// TIA Portal V16 export
// export: Created 2022-02-04T14:40:09.9916487Z, ExportSetting WithDefaults, DisplayName Totally Integrated Automation Portal, DisplayVersion V16 Update 1, DisplayName TIA Portal Version Control Interface, DisplayVersion V16, DisplayName TIA Portal Openness, DisplayVersion V16, DisplayName SINAMICS Startdrive Advanced, DisplayVersion V16 Update 5, DisplayName SINAMICS Startdrive G130, G150, S120, S150, SINAMICS MV, S210, DisplayVersion V16 Update 5, DisplayName SINAMICS Startdrive G110M, G120, G120C, G120D, G120P, G115D, DisplayVersion V16 Update 5, DisplayName STEP 7 Professional, DisplayVersion V16, DisplayName STEP 7 Safety, DisplayVersion V16, DisplayName WinCC Advanced, DisplayVersion V16, DisplayName SIMATIC Visualization Architect, DisplayVersion V16
FUNCTION_BLOCK "Беопасность"   // FB1, LAD
VERSION : 0.1
// stored: AutoNumber true, IsIECCheckEnabled false, UDAEnableTagReadback false
   VAR DB_SPECIFIC
      Trig61 : Bool;
      Trig62 : Bool;
      Trig63 : Bool;
      Trig64 : Bool;
      Trig65 : Bool;
      Trig66 : Bool;
      Trig67 : Bool;
      Trig69 : Bool;
      Trig68 : Bool;
      ProhibitionLoading : Bool := true;
      ProhibitionDefect : Bool := true;
      ProhibitionSorting : Bool := true;
      ProhibitionGasket : Bool := true;
   END_VAR
   VAR_TEMP
      AlarmReset : Bool;
   END_VAR
   VAR_TEMP   // added for the SCL form of the ladder/FBD networks
      _w1 : Bool;
      _w2 : Bool;
      _s5time1 : S5Time;
   END_VAR
BEGIN

REGION Network 1: Реле безопастности К10 ОСНОВНАЯ напряжение управления
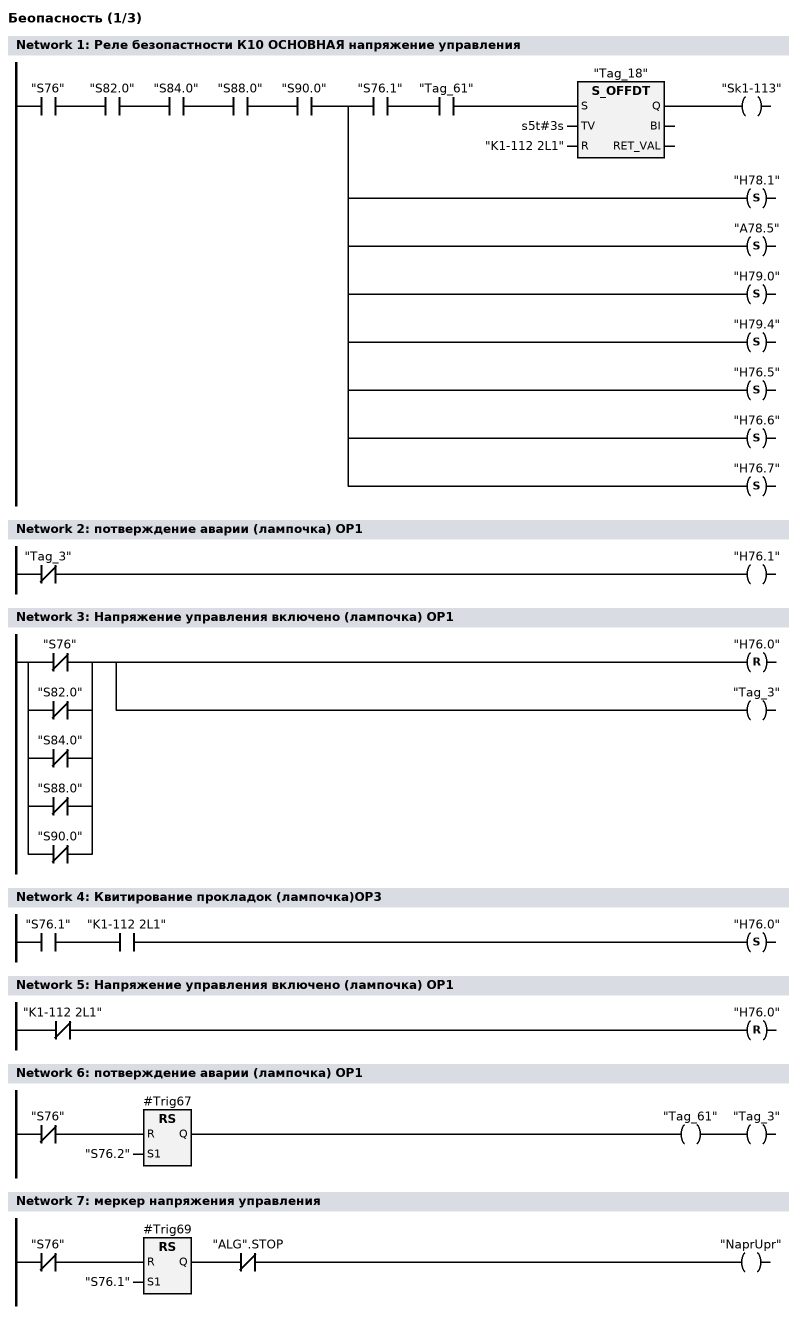
   RUNG wire#powerrail
      Contact( "S76" )
      Contact( "S82.0" )
      Contact( "S84.0" )
      Contact( "S88.0" )
      Contact( "S90.0" )
      wire#w1
      Contact( "S76.1" )
      Contact( "Tag_61" )
      S_OFFDT(T_NO := "Tag_18", TV := s5t#3s, R := "K1-112 2L1", BI =>, RET_VAL =>)
      Coil( "Sk1-113" )
   END_RUNG
   RUNG wire#w1
      S_Coil( "H78.1" )
   END_RUNG
   RUNG wire#w1
      S_Coil( "A78.5" )
   END_RUNG
   RUNG wire#w1
      S_Coil( "H79.0" )
   END_RUNG
   RUNG wire#w1
      S_Coil( "H79.4" )
   END_RUNG
   RUNG wire#w1
      S_Coil( "H76.5" )
   END_RUNG
   RUNG wire#w1
      S_Coil( "H76.6" )
   END_RUNG
   RUNG wire#w1
      S_Coil( "H76.7" )
   END_RUNG
   // the same network as SCL:
   #_w1 := "S76" AND "S82.0" AND "S84.0" AND "S88.0" AND "S90.0";
   #_s5time1 := S_OFFDT(T_NO := "Tag_18",
                        S := #_w1 AND "S76.1" AND "Tag_61",
                        TV := s5t#3s,
                        R := "K1-112 2L1",
                        Q => #_w2);
   "Sk1-113" := #_w2;
   IF #_w1 THEN
       "H78.1" := TRUE;
       "A78.5" := TRUE;
       "H79.0" := TRUE;
       "H79.4" := TRUE;
       "H76.5" := TRUE;
       "H76.6" := TRUE;
       "H76.7" := TRUE;
   END_IF;
END_REGION

REGION Network 2: потверждение аварии (лампочка) ОР1
   RUNG wire#powerrail
      I_Contact( "Tag_3" )
      Coil( "H76.1" )
   END_RUNG
   // the same network as SCL:
   "H76.1" := NOT "Tag_3";
END_REGION

REGION Network 3: Напряжение управления включено (лампочка) ОР1
   RUNG wire#powerrail
      I_Contact( "S76" )
      wire#w1
      R_Coil( "H76.0" )
   END_RUNG
   RUNG wire#powerrail
      I_Contact( "S82.0" )
   END_RUNG wire#w1
   RUNG wire#powerrail
      I_Contact( "S84.0" )
   END_RUNG wire#w1
   RUNG wire#powerrail
      I_Contact( "S88.0" )
   END_RUNG wire#w1
   RUNG wire#powerrail
      I_Contact( "S90.0" )
   END_RUNG wire#w1
   RUNG wire#w1
      Coil( "Tag_3" )
   END_RUNG
   // the same network as SCL:
   #_w1 := NOT "S76" OR NOT "S82.0" OR NOT "S84.0" OR NOT "S88.0" OR NOT "S90.0";
   IF #_w1 THEN "H76.0" := FALSE; END_IF;
   "Tag_3" := #_w1;
END_REGION

REGION Network 4: Квитирование прокладок (лампочка)ОР3
   RUNG wire#powerrail
      Contact( "S76.1" )
      Contact( "K1-112 2L1" )
      S_Coil( "H76.0" )
   END_RUNG
   // the same network as SCL:
   IF "S76.1" AND "K1-112 2L1" THEN "H76.0" := TRUE; END_IF;
END_REGION

REGION Network 5: Напряжение управления включено (лампочка) ОР1
   RUNG wire#powerrail
      I_Contact( "K1-112 2L1" )
      R_Coil( "H76.0" )
   END_RUNG
   // the same network as SCL:
   IF NOT "K1-112 2L1" THEN "H76.0" := FALSE; END_IF;
END_REGION

REGION Network 6: потверждение аварии (лампочка) ОР1
   RUNG wire#powerrail
      I_Contact( "S76" )
      S_RS(operand := #Trig67, s1 := "S76.2")
      Coil( "Tag_61" )
      Coil( "Tag_3" )
   END_RUNG
   // the same network as SCL:
   IF NOT "S76" THEN
       #Trig67 := FALSE;   // RS flip-flop
   END_IF;
   IF "S76.2" THEN #Trig67 := TRUE; END_IF;
   "Tag_61" := #Trig67;
   "Tag_3" := #Trig67;
END_REGION

REGION Network 7: меркер напряжения управления
   RUNG wire#powerrail
      I_Contact( "S76" )
      S_RS(operand := #Trig69, s1 := "S76.1")
      I_Contact( "ALG".STOP )
      Coil( "NaprUpr" )
   END_RUNG
   // the same network as SCL:
   IF NOT "S76" THEN
       #Trig69 := FALSE;   // RS flip-flop
   END_IF;
   IF "S76.1" THEN #Trig69 := TRUE; END_IF;
   "NaprUpr" := #Trig69 AND NOT "ALG".STOP;
END_REGION

REGION Network 8: Напряжение управления включено (лампочка) ОР1
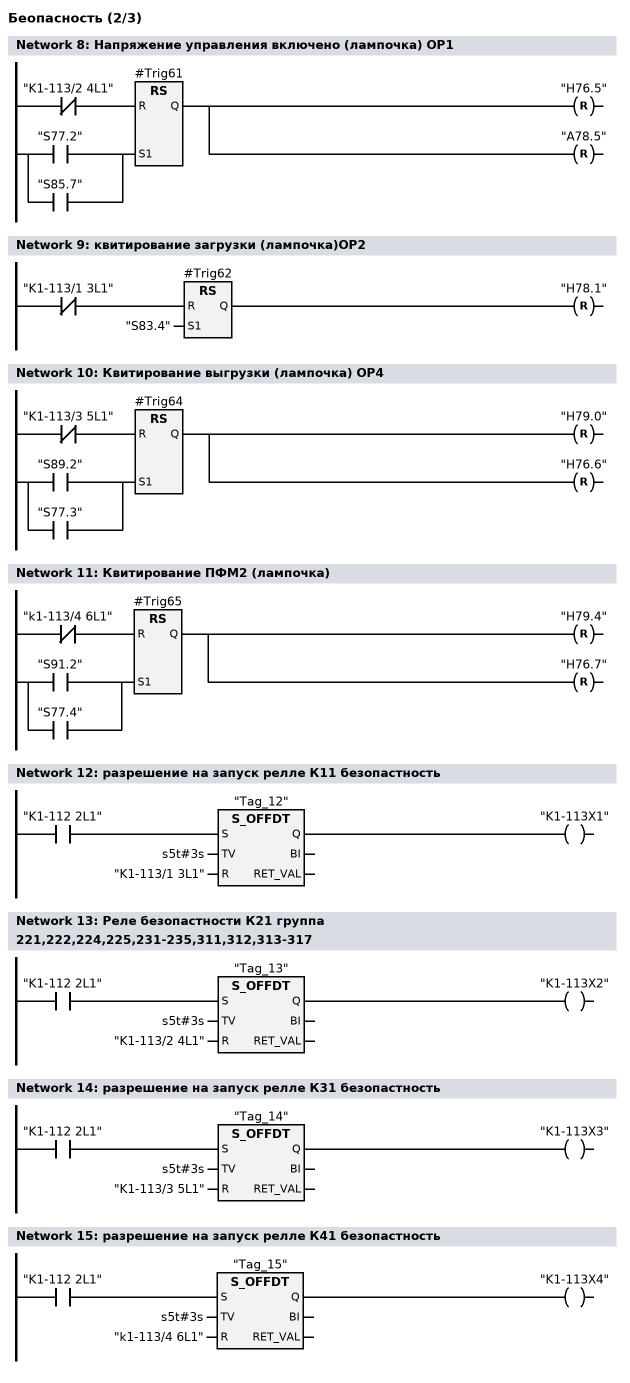
   RUNG wire#powerrail
      I_Contact( "K1-113/2 4L1" )
      S_RS(operand := #Trig61, s1 := wire#w1)
      wire#w2
      R_Coil( "H76.5" )
   END_RUNG
   RUNG wire#powerrail
      Contact( "S77.2" )
   END_RUNG wire#w1
   RUNG wire#powerrail
      Contact( "S85.7" )
   END_RUNG wire#w1
   RUNG wire#w2
      R_Coil( "A78.5" )
   END_RUNG
   // the same network as SCL:
   IF NOT "K1-113/2 4L1" THEN
       #Trig61 := FALSE;   // RS flip-flop
   END_IF;
   IF "S77.2" OR "S85.7" THEN #Trig61 := TRUE; END_IF;
   IF #Trig61 THEN
       "H76.5" := FALSE;
       "A78.5" := FALSE;
   END_IF;
END_REGION

REGION Network 9: квитирование загрузки (лампочка)ОР2
   RUNG wire#powerrail
      I_Contact( "K1-113/1 3L1" )
      S_RS(operand := #Trig62, s1 := "S83.4")
      R_Coil( "H78.1" )
   END_RUNG
   // the same network as SCL:
   IF NOT "K1-113/1 3L1" THEN
       #Trig62 := FALSE;   // RS flip-flop
   END_IF;
   IF "S83.4" THEN #Trig62 := TRUE; END_IF;
   IF #Trig62 THEN "H78.1" := FALSE; END_IF;
END_REGION

REGION Network 10: Квитирование выгрузки (лампочка) ОР4
   RUNG wire#powerrail
      I_Contact( "K1-113/3 5L1" )
      S_RS(operand := #Trig64, s1 := wire#w1)
      wire#w2
      R_Coil( "H79.0" )
   END_RUNG
   RUNG wire#powerrail
      Contact( "S89.2" )
   END_RUNG wire#w1
   RUNG wire#powerrail
      Contact( "S77.3" )
   END_RUNG wire#w1
   RUNG wire#w2
      R_Coil( "H76.6" )
   END_RUNG
   // the same network as SCL:
   IF NOT "K1-113/3 5L1" THEN
       #Trig64 := FALSE;   // RS flip-flop
   END_IF;
   IF "S89.2" OR "S77.3" THEN #Trig64 := TRUE; END_IF;
   IF #Trig64 THEN
       "H79.0" := FALSE;
       "H76.6" := FALSE;
   END_IF;
END_REGION

REGION Network 11: Квитирование ПФМ2 (лампочка)
   RUNG wire#powerrail
      I_Contact( "k1-113/4 6L1" )
      S_RS(operand := #Trig65, s1 := wire#w1)
      wire#w2
      R_Coil( "H79.4" )
   END_RUNG
   RUNG wire#powerrail
      Contact( "S91.2" )
   END_RUNG wire#w1
   RUNG wire#powerrail
      Contact( "S77.4" )
   END_RUNG wire#w1
   RUNG wire#w2
      R_Coil( "H76.7" )
   END_RUNG
   // the same network as SCL:
   IF NOT "k1-113/4 6L1" THEN
       #Trig65 := FALSE;   // RS flip-flop
   END_IF;
   IF "S91.2" OR "S77.4" THEN #Trig65 := TRUE; END_IF;
   IF #Trig65 THEN
       "H79.4" := FALSE;
       "H76.7" := FALSE;
   END_IF;
END_REGION

REGION Network 12: разрешение на запуск релле К11 безопастность
   RUNG wire#powerrail
      Contact( "K1-112 2L1" )
      S_OFFDT(T_NO := "Tag_12", TV := s5t#3s, R := "K1-113/1 3L1", BI =>, RET_VAL =>)
      Coil( "K1-113X1" )
   END_RUNG
   // the same network as SCL:
   #_s5time1 := S_OFFDT(T_NO := "Tag_12", S := "K1-112 2L1", TV := s5t#3s, R := "K1-113/1 3L1", Q => #_w1);
   "K1-113X1" := #_w1;
END_REGION

REGION Network 13: Реле безопастности К21 группа 221,222,224,225,231-235,311,312,313-317
   RUNG wire#powerrail
      Contact( "K1-112 2L1" )
      S_OFFDT(T_NO := "Tag_13", TV := s5t#3s, R := "K1-113/2 4L1", BI =>, RET_VAL =>)
      Coil( "K1-113X2" )
   END_RUNG
   // the same network as SCL:
   #_s5time1 := S_OFFDT(T_NO := "Tag_13", S := "K1-112 2L1", TV := s5t#3s, R := "K1-113/2 4L1", Q => #_w1);
   "K1-113X2" := #_w1;
END_REGION

REGION Network 14: разрешение на запуск релле К31 безопастность
   RUNG wire#powerrail
      Contact( "K1-112 2L1" )
      S_OFFDT(T_NO := "Tag_14", TV := s5t#3s, R := "K1-113/3 5L1", BI =>, RET_VAL =>)
      Coil( "K1-113X3" )
   END_RUNG
   // the same network as SCL:
   #_s5time1 := S_OFFDT(T_NO := "Tag_14", S := "K1-112 2L1", TV := s5t#3s, R := "K1-113/3 5L1", Q => #_w1);
   "K1-113X3" := #_w1;
END_REGION

REGION Network 15: разрешение на запуск релле К41 безопастность
   RUNG wire#powerrail
      Contact( "K1-112 2L1" )
      S_OFFDT(T_NO := "Tag_15", TV := s5t#3s, R := "k1-113/4 6L1", BI =>, RET_VAL =>)
      Coil( "K1-113X4" )
   END_RUNG
   // the same network as SCL:
   #_s5time1 := S_OFFDT(T_NO := "Tag_15", S := "K1-112 2L1", TV := s5t#3s, R := "k1-113/4 6L1", Q => #_w1);
   "K1-113X4" := #_w1;
END_REGION

REGION Network 16: Сирена начало работы
   // сирена горит 5 секунд и дает разрешение на включение нужного режима
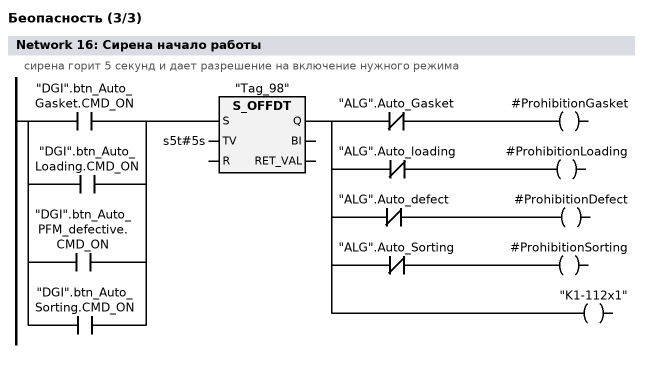
   RUNG wire#powerrail
      Contact( "DGI".btn_Auto_Gasket.CMD_ON )
      wire#w1
      S_OFFDT(T_NO := "Tag_98", TV := s5t#5s, R :=, BI =>, RET_VAL =>)
      wire#w2
      I_Contact( "ALG".Auto_Gasket )
      Coil( #ProhibitionGasket )
   END_RUNG
   RUNG wire#powerrail
      Contact( "DGI".btn_Auto_Loading.CMD_ON )
   END_RUNG wire#w1
   RUNG wire#powerrail
      Contact( "DGI".btn_Auto_PFM_defective.CMD_ON )
   END_RUNG wire#w1
   RUNG wire#powerrail
      Contact( "DGI".btn_Auto_Sorting.CMD_ON )
   END_RUNG wire#w1
   RUNG wire#w2
      I_Contact( "ALG".Auto_loading )
      Coil( #ProhibitionLoading )
   END_RUNG
   RUNG wire#w2
      I_Contact( "ALG".Auto_defect )
      Coil( #ProhibitionDefect )
   END_RUNG
   RUNG wire#w2
      I_Contact( "ALG".Auto_Sorting )
      Coil( #ProhibitionSorting )
   END_RUNG
   RUNG wire#w2
      Coil( "K1-112x1" )
   END_RUNG
   // the same network as SCL:
   #_s5time1 := S_OFFDT(T_NO := "Tag_98",
                        S := "DGI".btn_Auto_Gasket.CMD_ON OR "DGI".btn_Auto_Loading.CMD_ON OR "DGI".btn_Auto_PFM_defective.CMD_ON OR "DGI".btn_Auto_Sorting.CMD_ON,
                        TV := s5t#5s,
                        Q => #_w1);
   #ProhibitionGasket := #_w1 AND NOT "ALG".Auto_Gasket;
   #ProhibitionLoading := #_w1 AND NOT "ALG".Auto_loading;
   #ProhibitionDefect := #_w1 AND NOT "ALG".Auto_defect;
   #ProhibitionSorting := #_w1 AND NOT "ALG".Auto_Sorting;
   "K1-112x1" := #_w1;
END_REGION
END_FUNCTION_BLOCK
